(* CoDeSys 2.3 export: EvtCh8Tick32Int32.EXP *)

(* POU core/evt/EvtCh8Tick32Int32, ST *)
FUNCTION EvtCh8Tick32Int32 : BOOL
VAR_INPUT
    Channel: BYTE;
    Tick: UDINT;
    Value: DINT;
END_VAR
VAR_IN_OUT
    Handle: LogBufferHandle;
END_VAR
VAR
    i: DINT;
    p1: POINTER TO BYTE;
    p2: POINTER TO BYTE;
    p3: POINTER TO UDINT;
    p4: POINTER TO DINT;
END_VAR
i := GetNextWritePointer(17, Handle.BufferWritePointer, Handle.BufferReadPointer, Handle.BufferSize, Handle.BufferOverflow);
IF i >= 0 THEN

    p1 := Handle.BufferAddress + DINT_TO_DWORD(i);
    p1^ := START_FLAG;

    p1 := p1 + 1;
    p1^ := Handle.MagicByte;

    p1 := p1 + 1;
    p1^ := EVT_CH8_TICK32_INT32;

    p1 := p1 + 1;
    p1^ := Channel;

    p3 := p1 + 1;
    p3^ := Tick;

    p4 := p1 + 5;
    p4^ := Value;

    p1 := p1 + 9;
    p1^ := END_FLAG;

    Handle.BufferWritePointer := DWORD_TO_DINT(p1 - Handle.BufferAddress);

ELSE
    EvtFull(Handle);
END_IF
END_FUNCTION
